// TIA Portal V16 export
// export: Created 2024-09-05T17:40:14.0556327Z, ExportSetting WithDefaults, DisplayName Totally Integrated Automation Portal, DisplayVersion V16 Update 6, DisplayName TIA Portal Version Control Interface, DisplayVersion V16 Update 2, DisplayName TIA Portal Openness, DisplayVersion V16 Update 6, DisplayName STEP 7 Professional, DisplayVersion V16 Update 6, DisplayName STEP 7 Safety, DisplayVersion V16, DisplayName WinCC Advanced, DisplayVersion V16 Update 6
TYPE "UDT_CognexReaders"
// stored: IsFailsafeCompliant false
   STRUCT
      HW : Struct
         In : Struct
            AcquisitionStatus : HW_MODULE;
            ResultsStatus : HW_MODULE;
            SoftEventControl : HW_MODULE;
            ResultData : HW_MODULE;
         END_STRUCT;
         Out : Struct
            AcquisitionControl : HW_MODULE;
            ResultsControl : HW_MODULE;
            SoftEventControl : HW_MODULE;
            UserData : HW_MODULE;
         END_STRUCT;
      END_STRUCT;
      ST : Struct
         RequestNewTrigger : Bool;
         ResultPending : Bool;
         LatestResults : Struct
            ID : Int;
            Flags : Int;
            Lenght : Int;
            Data : Array[1..64] of Byte;
         END_STRUCT;
      END_STRUCT;
   END_STRUCT;
END_TYPE
